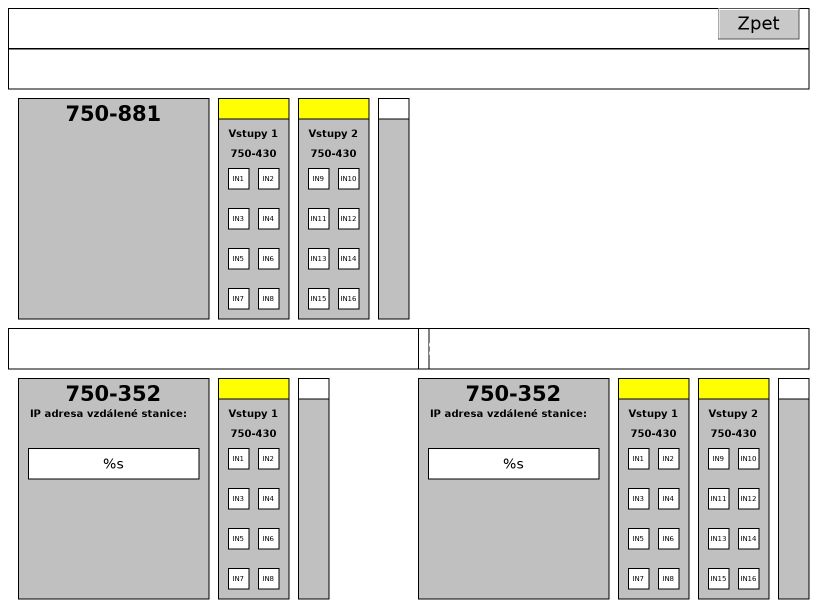
[picture p24: Servis (HMI screen)]
rectangle at (0,0)-(801,41): text "SERVIS"
rectangle at (220,160)-(241,181): text "IN1"; alarm colour if IN1
rectangle at (210,110)-(281,141): text "Vstupy 1"
rectangle at (250,160)-(271,181): text "IN2"; alarm colour if IN2
rectangle at (210,130)-(281,161): text "750-430"
rectangle at (10,90)-(201,121): text "750-881"
rectangle at (220,200)-(241,221): text "IN3"; alarm colour if IN3
rectangle at (250,200)-(271,221): text "IN4"; alarm colour if IN4
rectangle at (220,240)-(241,261): text "IN5"; alarm colour if IN5
rectangle at (250,240)-(271,261): text "IN6"; alarm colour if IN6
rectangle at (220,280)-(241,301): text "IN7"; alarm colour if IN7
rectangle at (250,280)-(271,301): text "IN8"; alarm colour if IN8
rectangle at (300,160)-(321,181): text "IN9"; alarm colour if IN9
rectangle at (290,110)-(361,141): text "Vstupy 2"
rectangle at (330,160)-(351,181): text "IN10"; alarm colour if VzdalenyVstup2
rectangle at (290,130)-(361,161): text "750-430"
rectangle at (300,200)-(321,221): text "IN11"; alarm colour if IN11
rectangle at (330,200)-(351,221): text "IN12"; alarm colour if IN12
rectangle at (300,240)-(321,261): text "IN13"; alarm colour if IN13
rectangle at (330,240)-(351,261): text "IN14"; alarm colour if IN14
rectangle at (300,280)-(321,301): text "IN15"; alarm colour if IN15
rectangle at (330,280)-(351,301): text "IN16"; alarm colour if IN16
rectangle at (220,440)-(241,461): text "IN1"; alarm colour if Host1IN1
rectangle at (210,390)-(281,421): text "Vstupy 1"
rectangle at (250,440)-(271,461): text "IN2"; alarm colour if Host1IN2
rectangle at (210,410)-(281,441): text "750-430"
rectangle at (10,370)-(201,401): text "750-352"
rectangle at (10,390)-(191,421): text "IP adresa vzdálené stanice:"
rectangle at (20,440)-(191,471): text "%s"; shows IPHost1
rectangle at (220,480)-(241,501): text "IN3"; alarm colour if Host1IN3
rectangle at (250,480)-(271,501): text "IN4"; alarm colour if Host1IN4
rectangle at (220,520)-(241,541): text "IN5"; alarm colour if Host1IN5
rectangle at (250,520)-(271,541): text "IN6"; alarm colour if Host1IN6
rectangle at (220,560)-(241,581): text "IN7"; alarm colour if Host1IN7
rectangle at (250,560)-(271,581): text "IN8"; alarm colour if Host1IN8
rectangle at (620,440)-(641,461): text "IN1"; alarm colour if Host2IN1
rectangle at (610,390)-(681,421): text "Vstupy 1"
rectangle at (650,440)-(671,461): text "IN2"; alarm colour if Host2IN2
rectangle at (610,410)-(681,441): text "750-430"
rectangle at (410,370)-(601,401): text "750-352"
rectangle at (410,390)-(591,421): text "IP adresa vzdálené stanice:"
rectangle at (420,440)-(591,471): text "%s"; shows IPHost2
rectangle at (620,480)-(641,501): text "IN3"; alarm colour if Host2IN3
rectangle at (650,480)-(671,501): text "IN4"; alarm colour if Host2IN4
rectangle at (620,520)-(641,541): text "IN5"; alarm colour if Host2IN5
rectangle at (650,520)-(671,541): text "IN6"; alarm colour if Host2IN6
rectangle at (620,560)-(641,581): text "IN7"; alarm colour if Host2IN7
rectangle at (650,560)-(671,581): text "IN8"; alarm colour if Host2IN8
rectangle at (0,40)-(801,81): text "SLEVARNA AL OJS I"
rectangle at (0,320)-(421,361): text "SLEVARNA AL OJS II"
rectangle at (410,320)-(801,361): text "SLEVARNA AL OJS III"
button at (710,0)-(791,31): text "Zpet"; opens plc_vizu
rectangle at (700,440)-(721,461): text "IN9"; alarm colour if Host2IN9
rectangle at (690,390)-(761,421): text "Vstupy 2"
rectangle at (730,440)-(751,461): text "IN10"; alarm colour if Host2IN10
rectangle at (690,410)-(761,441): text "750-430"
rectangle at (700,480)-(721,501): text "IN11"; alarm colour if Host2IN11
rectangle at (730,480)-(751,501): text "IN12"; alarm colour if Host2IN12
rectangle at (700,520)-(721,541): text "IN13"; alarm colour if Host2IN13
rectangle at (730,520)-(751,541): text "IN14"; alarm colour if Host2IN14
rectangle at (700,560)-(721,581): text "IN15"; alarm colour if Host2IN15
rectangle at (730,560)-(751,581): text "IN16"; alarm colour if Host2IN16
19 more shapes without text or variables
*)

(* Visualisation Slitina
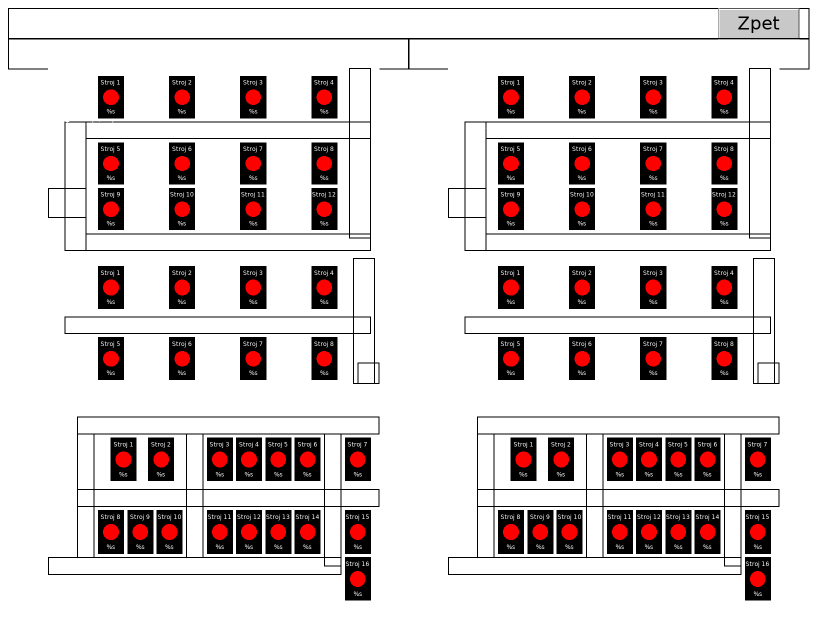
rectangle at (0,0)-(801,31): text "SLITINY"
button at (710,0)-(791,31): text "Zpet"; opens plc_vizu
rectangle at (0,30)-(401,61): text "%s"; shows PLC_PRG.Slitina[1]
rectangle at (400,30)-(801,61): text "%s"; shows PLC_PRG.Slitina[1]
embedded screen at (40,60)-(371,251): OJS_I_FS1x
embedded screen at (40,250)-(371,401): OJS_II_FS1x
embedded screen at (40,400)-(371,601): OJS_III_FS1x
embedded screen at (440,60)-(771,251): OJS_I_FS2x
embedded screen at (440,250)-(771,401): OJS_II_FS2x
embedded screen at (440,400)-(771,601): OJS_III_FS2x
*)
